FUNCTION F_RotationsPerMinute : UDINT
VAR_INPUT
END_VAR
VAR
END_VAR

//asd

END_FUNCTION

(* stored: Version 1.1.0.1, ProductVersion 3.1.4024.10
   POU F_RotationsPerMinute: Id {26c608cd-7a09-42cc-88c8-6cdabbc35695}, SpecialFunc None *)
